(* Logix 5000 project; controller PBS_Perfusion vendor 1 type 14 code 217 rev 32.14; software revision 32.03; part 25 of 27 *)
(* tags used below, declared in another part *)
   AIC703 : P_AInAdv;   // BRX DO PV
   AT701 : P_AInAdv;   // DO Transmitter
   AT702 : P_AInAdv;   // pH Transmitter
   BRX_Comm_Toggle : BOOL;
   BRX_Data : PBSdata_UDT;
   Brx_heartbeat_Alarm : BOOL;
   Brx_Heartbeat_Alarm_Reset : BOOL;
   BRX_Heartbeat_Fail : TIMER;
   BRX_HiAdj : BOOL;   // BRX HI adj in progress
   BRX_HiAdjEnable : BOOL;
   BRX_HiAdjTimer : TIMER;
   BRX_HiadjTimeSP : REAL;
   BRX_HiSP : REAL;
   BRX_LoAdj : BOOL;   // BRX Lo Adj in progress
   BRX_LoAdjEnable : BOOL;
   BRX_LoAdjTimer : TIMER;
   BRX_LoadjTimeSP : REAL;
   BRX_LoSP : REAL;
   ConditionedMedia_Initialize : BOOL;
   ConditionedMedia_Scaler : SCALE;
   CondMed_AdjustInProgress : BOOL;
   EStop : P_DIn;
   Heater_Output : P_AOut;   // Heating blanket AO
   Heater_Output_intlk : P_Intlk;
   Json_Alarm : BOOL;
   LIT801 : P_AInAdv;   // Level Value From BRX
   MCV_HiAdj : BOOL;   // MCV hi adjust active
   MCV_HiAdjEnable : BOOL;
   MCV_HiAdjTimer : TIMER;
   MCV_HiAdjTimeSP : REAL;
   MCV_HiSP : REAL;
   ONS : DINT[3];
   P101 : P_VSD;   // Feed Pump
   P101_Alarm_Reset : AMP_Alarm_Reset;
   P101_Cal : Pump_Cal;
   P101_Cal_Constant : REAL;
   P101_Crash_Stop : AMP_Crash_Stop;
   P101_Dose_Running : BOOL;
   P101_Dose_Speed_mlmin : REAL;
   P101_Enable : AMP_Motor_Enable;
   P101_FaultCodeList : P_DescList[1];
   P101_Input_Assembly : AMP_Input_Assembly_v2;
   P101_Input_Assembly_Instance : AMP_Input_Assembly;
   P101_intlk : P_Intlk;
   P101_Jog_Move : AMP_Jog_Move;
   P101_Relative_Move : AMP_Relative_Move;
   P101_Status_Code : AMP_Status_Code;
   P101_Update_Jog_Speed : AMP_Update_Jog_Speed;
   P101Fault : BOOL;
   P101Fault_Output : BOOL;
   P102 : P_VSD;   // Media Pump
   P102_Alarm_Reset : AMP_Alarm_Reset;
   P102_Cal : Pump_Cal;
   P102_Cal_Constant : REAL;
   P102_Crash_Stop : AMP_Crash_Stop;
   P102_Enable : AMP_Motor_Enable;
   P102_FaultCodeList : P_DescList[1];
   P102_Input_Assembly : AMP_Input_Assembly_v2;
   P102_Input_Assembly_Instance : AMP_Input_Assembly;
   P102_intlk : P_Intlk;
   P102_Jog_Move : AMP_Jog_Move;
   P102_Relative_Move : AMP_Relative_Move;
   P102_Status_Code : AMP_Status_Code;
   P102_Update_Jog_Speed : AMP_Update_Jog_Speed;
   P103 : P_VSD;   // Conditioned Media Addition Pump
   P103_Alarm_Reset : AMP_Alarm_Reset;
   P103_Cal : Pump_Cal;
   P103_Cal_Constant : REAL;
   P103_Crash_Stop : AMP_Crash_Stop;
   P103_Enable : AMP_Motor_Enable;
   P103_FaultCodeList : P_DescList[1];
   P103_Input_Assembly : AMP_Input_Assembly_v2;
   P103_Input_Assembly_Instance : AMP_Input_Assembly;
   P103_intlk : P_Intlk;
   P103_Jog_Move : AMP_Jog_Move;
   P103_Relative_Move : AMP_Relative_Move;
   P103_Status_Code : AMP_Status_Code;
   P103_Update_Jog_Speed : AMP_Update_Jog_Speed;
   P104 : P_VSD;   // Recirculation Pump
   P104_Alarm_Reset : AMP_Alarm_Reset;
   P104_Cal : Pump_Cal;
   P104_Cal_Constant : REAL;
   P104_Crash_Stop : AMP_Crash_Stop;
   P104_Enable : AMP_Motor_Enable;
   P104_FaultCodeList : P_DescList[1];
   P104_Input_Assembly : AMP_Input_Assembly_v2;
   P104_Input_Assembly_Instance : AMP_Input_Assembly;
   p104_intlk : P_Intlk;
   P104_Jog_Move : AMP_Jog_Move;
   P104_Relative_Move : AMP_Relative_Move;
   P104_Status_Code : AMP_Status_Code;
   P104_Update_Jog_Speed : AMP_Update_Jog_Speed;
   P105 : P_VSD;   // Spent Media Pump
   P105_FaultCodeList : P_DescList[1];
   P105_intlk : P_Intlk;
   Recirc_HiSP1 : REAL;   // BRX Hi recirc hi speed modifier
   Recirc_LoSP1 : REAL;   // MCV Hi recirc lo speed modifier
   Recirc_LoSP2 : REAL;   // BRX Lo recirc lo speed modifier
   SIC401 : P_VSD;   // Agitator
   SIC401_FaultCodeList : P_DescList[1];   // made for agaitor p_VSD block
   SIC401_intlk : P_Intlk;
   Temp_Limit_Adm : REAL;
   Temp_Scaler : SCALE;
   Test_Temp_Raw : REAL;
   TT700 : P_AInAdv;   // Temperature Transmitter
   WT701 : P_AInAdv;   // Media Scale
   WT702 : P_AInAdv;   // MCV Weight
   WT703 : P_AInAdv;   // Spent Media/Harvest Scale

PROGRAM CM_PBS   (* main routine Main *)
VAR
   BOR_01 : FBD_BOOLEAN_OR;
   SEL_01 : SELECT := (In2 := 200.0);
   TOT_01 : TOTALIZER := (Gain := 1.0, RTSTime := 1);
   TOT_02 : TOTALIZER := (Gain := 1.0, RTSTime := 1);
END_VAR

ROUTINE Brx_Comms   (* ladder *)
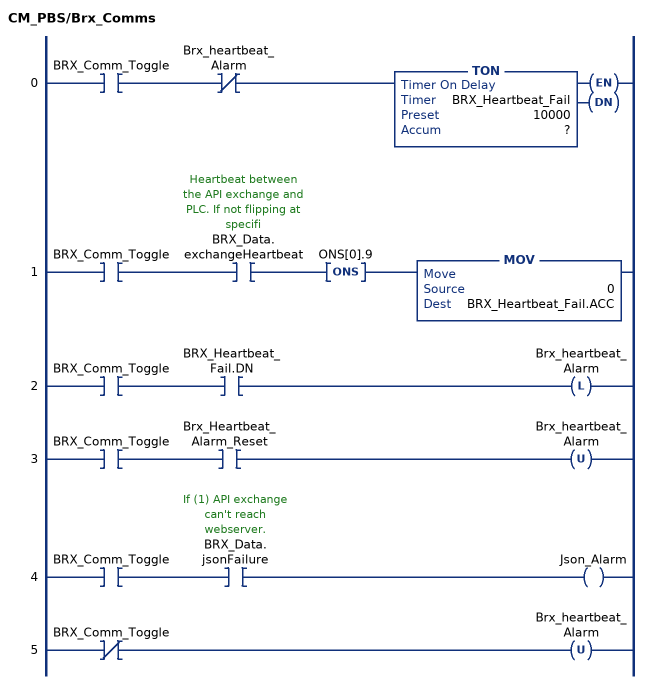
   0: XIC(BRX_Comm_Toggle)XIO(Brx_heartbeat_Alarm)TON(BRX_Heartbeat_Fail,?,?);
   1: XIC(BRX_Comm_Toggle)XIC(BRX_Data.exchangeHeartbeat)ONS(ONS[0].9)MOV(0,BRX_Heartbeat_Fail.ACC);
   2: XIC(BRX_Comm_Toggle)XIC(BRX_Heartbeat_Fail.DN)OTL(Brx_heartbeat_Alarm);
   3: XIC(BRX_Comm_Toggle)XIC(Brx_Heartbeat_Alarm_Reset)OTU(Brx_heartbeat_Alarm);
   4: XIC(BRX_Comm_Toggle)XIC(BRX_Data.jsonFailure)OTE(Json_Alarm);
   5: XIO(BRX_Comm_Toggle)OTU(Brx_heartbeat_Alarm);
END_ROUTINE

ROUTINE CM_Agitator   (* ladder *)
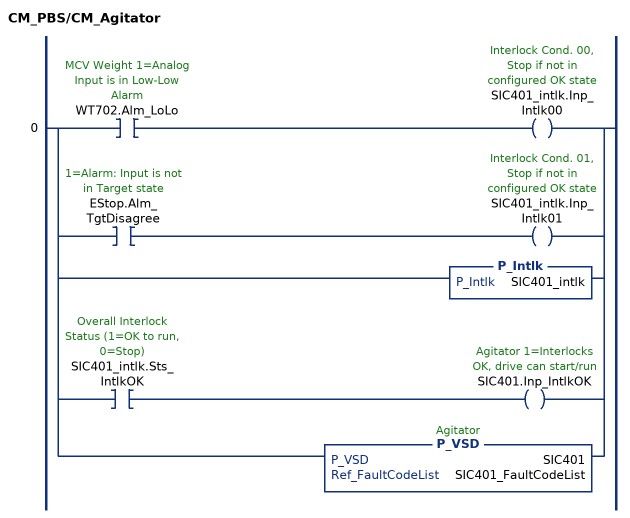
   0: [[XIC(WT702.Alm_LoLo) OTE(SIC401_intlk.Inp_Intlk00) ,XIC(EStop.Alm_TgtDisagree) OTE(SIC401_intlk.Inp_Intlk01) ,P_Intlk(SIC401_intlk) ,XIC(SIC401_intlk.Sts_IntlkOK) OTE(SIC401.Inp_IntlkOK) ] ,P_VSD(SIC401,SIC401_FaultCodeList) ];
END_ROUTINE

ROUTINE CM_AI   (* ladder *)
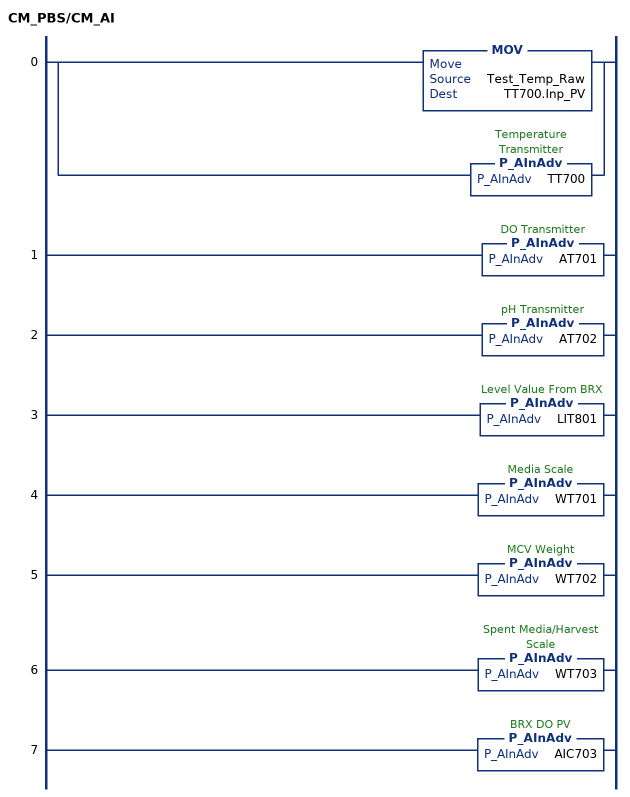
   0: [MOV(Test_Temp_Raw,TT700.Inp_PV) ,P_AInAdv(TT700) ];
   1: P_AInAdv(AT701);
   2: P_AInAdv(AT702);
   3: P_AInAdv(LIT801);
   4: P_AInAdv(WT701);
   5: P_AInAdv(WT702);
   6: P_AInAdv(WT703);
   7: P_AInAdv(AIC703);
END_ROUTINE

ROUTINE CM_AO   (* ladder *)
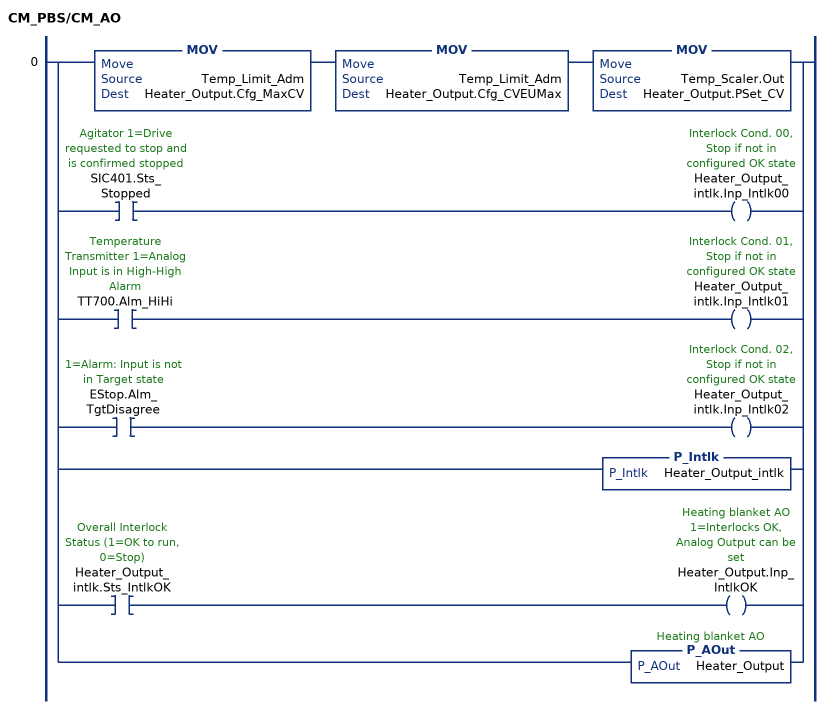
   0: [MOV(Temp_Limit_Adm,Heater_Output.Cfg_MaxCV) MOV(Temp_Limit_Adm,Heater_Output.Cfg_CVEUMax) MOV(Temp_Scaler.Out,Heater_Output.PSet_CV) ,[XIC(SIC401.Sts_Stopped) OTE(Heater_Output_intlk.Inp_Intlk00) ,XIC(TT700.Alm_HiHi) OTE(Heater_Output_intlk.Inp_Intlk01) ,XIC(EStop.Alm_TgtDisagree) OTE(Heater_Output_intlk.Inp_Intlk02) ,P_Intlk(Heater_Output_intlk) ,XIC(Heater_Output_intlk.Sts_IntlkOK) OTE(Heater_Output.Inp_IntlkOK) ] ,P_AOut(Heater_Output) ];
END_ROUTINE

ROUTINE CM_DI   (* ladder *)
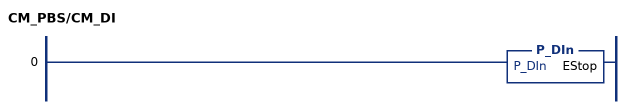
   0: P_DIn(EStop);
END_ROUTINE

ROUTINE CM_DO   (* ladder *)
END_ROUTINE

ROUTINE CM_Pumps   (* ladder *)
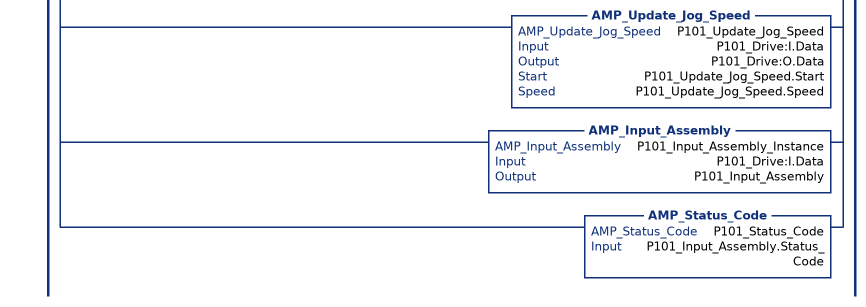
   0: [XIC(P101Fault) OTE(P101Fault_Output) ,[XIC(LIT801.Alm_HiHi) OTE(P101_intlk.Inp_Intlk00) ,XIC(WT701.Alm_LoLo) OTE(P101_intlk.Inp_Intlk01) ,XIC(EStop.Alm_TgtDisagree) OTE(P101_intlk.Inp_Intlk02) ,P_Intlk(P101_intlk) ,XIC(P101_intlk.Sts_IntlkOK) OTE(P101.Inp_IntlkOK) ] ,[P_VSD(P101,P101_FaultCodeList) ,XIC(P101.Sts_StartingFwd) OTL(P101_Jog_Move.Start) ,XIC(P101.Sts_StoppingFwd) OTL(P101_Crash_Stop.Stop) ,XIC(P101_Status_Code.Moving) OTU(P101_Jog_Move.Start) ,XIO(P101_Status_Code.Moving) OTU(P101_Crash_Stop.Stop) ,CPT(P101_Jog_Move.Speed,P101.Val_SpeedRef/ ( P101_Cal_Constant * 60)) ,NEQ(P101_Update_Jog_Speed.Speed,P101_Jog_Move.Speed) ONS(ONS[0].5) MOV(P101_Jog_Move.Speed,P101_Update_Jog_Speed.Speed) OTE(P101_Update_Jog_Speed.Start) ] ,AFI() Pump_Cal(P101_Cal,P101.Sts_RunningFwd,P101.PCmd_Prog,P101.Cfg_SpeedRefEUMin,P101.Cfg_SpeedRefEUMax,P101.Cfg_SpeedFdbkEUMin,P101.Cfg_SpeedFdbkEUMax,P101.Cfg_MinSpdRef,P101.Cfg_MaxSpdRef,P101.PSet_SpeedRef,P101.PCmd_StartFwd,P101.Sts_Prog,P101.PCmd_Stop) ,AMP_Motor_Enable(P101_Enable,P101_Drive:I.Data,P101_Drive:O.Data,P101_Enable.Enable) ,AMP_Alarm_Reset(P101_Alarm_Reset,P101_Drive:I.Data,P101_Drive:O.Data,P101_Alarm_Reset.Reset) ,AMP_Jog_Move(P101_Jog_Move,P101_Drive:I.Data,P101_Drive:O.Data,P101_Jog_Move.Start,P101_Jog_Move.Speed,P101_Jog_Move.Acc,P101_Jog_Move.Dec) ,AMP_Crash_Stop(P101_Crash_Stop,P101_Drive:I.Data,P101_Drive:O.Data,P101_Crash_Stop.Stop) ,AMP_Relative_Move(P101_Relative_Move,P101_Drive:I.Data,P101_Drive:O.Data,P101_Relative_Move.Start,P101_Relative_Move.Distance,P101_Relative_Move.Speed,P101_Relative_Move.Acc,P101_Relative_Move.Dec) ,AMP_Update_Jog_Speed(P101_Update_Jog_Speed,P101_Drive:I.Data,P101_Drive:O.Data,P101_Update_Jog_Speed.Start,P101_Update_Jog_Speed.Speed) ,AMP_Input_Assembly(P101_Input_Assembly_Instance,P101_Drive:I.Data,P101_Input_Assembly) ,AMP_Status_Code(P101_Status_Code,P101_Input_Assembly.Status_Code) ];
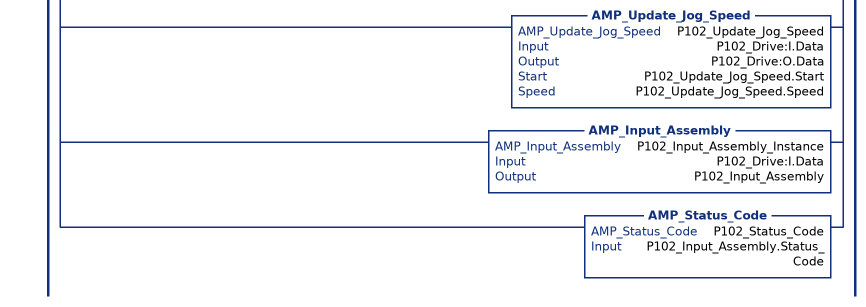
   1: [[XIC(WT702.Alm_HiHi) OTE(P102_intlk.Inp_Intlk00) ,XIC(WT701.Alm_LoLo) OTE(P102_intlk.Inp_Intlk01) ,XIC(EStop.Alm_TgtDisagree) OTE(P102_intlk.Inp_Intlk02) ,P_Intlk(P102_intlk) ,XIC(P102_intlk.Sts_IntlkOK) OTE(P102.Inp_IntlkOK) ] ,[P_VSD(P102,P102_FaultCodeList) ,XIC(P102.Sts_StartingFwd) OTL(P102_Jog_Move.Start) ,XIC(P102.Sts_StoppingFwd) OTL(P102_Crash_Stop.Stop) ,XIC(P102_Status_Code.Moving) OTU(P102_Jog_Move.Start) ,XIO(P102_Status_Code.Moving) OTU(P102_Crash_Stop.Stop) ,CPT(P102_Jog_Move.Speed,P102.Val_SpeedRef/ ( P102_Cal_Constant * 60)) ,NEQ(P102_Update_Jog_Speed.Speed,P102_Jog_Move.Speed) ONS(ONS[0].5) MOV(P102_Jog_Move.Speed,P102_Update_Jog_Speed.Speed) OTE(P102_Update_Jog_Speed.Start) ] ,AFI() Pump_Cal(P102_Cal,P102.Sts_RunningFwd,P102.PCmd_Prog,P102.Cfg_SpeedRefEUMin,P102.Cfg_SpeedRefEUMax,P102.Cfg_SpeedFdbkEUMin,P102.Cfg_SpeedFdbkEUMax,P102.Cfg_MinSpdRef,P102.Cfg_MaxSpdRef,P102.PSet_SpeedRef,P102.PCmd_StartFwd,P102.Sts_Prog,P102.PCmd_Stop) ,AMP_Motor_Enable(P102_Enable,P102_Drive:I.Data,P102_Drive:O.Data,P102_Enable.Enable) ,AMP_Alarm_Reset(P102_Alarm_Reset,P102_Drive:I.Data,P102_Drive:O.Data,P102_Alarm_Reset.Reset) ,AMP_Jog_Move(P102_Jog_Move,P102_Drive:I.Data,P102_Drive:O.Data,P102_Jog_Move.Start,P102_Jog_Move.Speed,P102_Jog_Move.Acc,P102_Jog_Move.Dec) ,AMP_Crash_Stop(P102_Crash_Stop,P102_Drive:I.Data,P102_Drive:O.Data,P102_Crash_Stop.Stop) ,AMP_Relative_Move(P102_Relative_Move,P102_Drive:I.Data,P102_Drive:O.Data,P102_Relative_Move.Start,P102_Relative_Move.Distance,P102_Relative_Move.Speed,P102_Relative_Move.Acc,P102_Relative_Move.Dec) ,AMP_Update_Jog_Speed(P102_Update_Jog_Speed,P102_Drive:I.Data,P102_Drive:O.Data,P102_Update_Jog_Speed.Start,P102_Update_Jog_Speed.Speed) ,AMP_Input_Assembly(P102_Input_Assembly_Instance,P102_Drive:I.Data,P102_Input_Assembly) ,AMP_Status_Code(P102_Status_Code,P102_Input_Assembly.Status_Code) ];
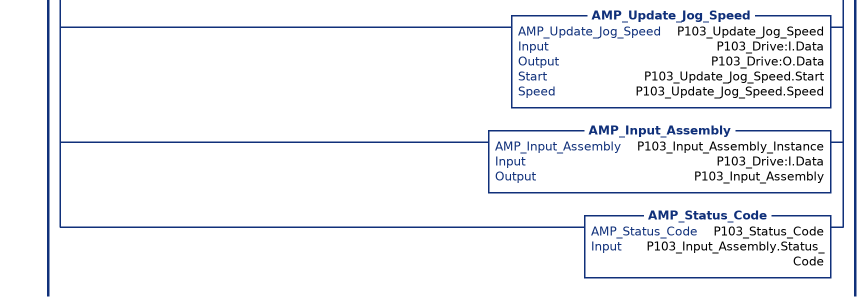
   2: [[XIC(LIT801.Alm_HiHi) OTE(P103_intlk.Inp_Intlk00) ,XIC(WT702.Alm_LoLo) OTE(P103_intlk.Inp_Intlk01) ,XIC(EStop.Alm_TgtDisagree) OTE(P103_intlk.Inp_Intlk02) ,P_Intlk(P103_intlk) ,XIC(P103_intlk.Sts_IntlkOK) OTE(P103.Inp_IntlkOK) ] ,[P_VSD(P103,P103_FaultCodeList) ,XIC(P103.Sts_StartingFwd) OTL(P103_Jog_Move.Start) ,XIC(P103.Sts_StoppingFwd) OTL(P103_Crash_Stop.Stop) ,XIC(P103_Status_Code.Moving) OTU(P103_Jog_Move.Start) ,XIO(P103_Status_Code.Moving) OTU(P103_Crash_Stop.Stop) ,CPT(P103_Jog_Move.Speed,P103.Val_SpeedRef/ ( P103_Cal_Constant * 60)) ,NEQ(P103_Update_Jog_Speed.Speed,P103_Jog_Move.Speed) ONS(ONS[0].5) MOV(P103_Jog_Move.Speed,P103_Update_Jog_Speed.Speed) OTE(P102_Update_Jog_Speed.Start) ] ,AFI() Pump_Cal(P103_Cal,P103.Sts_RunningFwd,P103.PCmd_Prog,P103.Cfg_SpeedRefEUMin,P103.Cfg_SpeedRefEUMax,P103.Cfg_SpeedFdbkEUMin,P103.Cfg_SpeedFdbkEUMax,P103.Cfg_MinSpdRef,P103.Cfg_MaxSpdRef,P103.PSet_SpeedRef,P103.PCmd_StartFwd,P103.Sts_Prog,P103.PCmd_Stop) ,AMP_Motor_Enable(P103_Enable,P103_Drive:I.Data,P103_Drive:O.Data,P103_Enable.Enable) ,AMP_Alarm_Reset(P103_Alarm_Reset,P103_Drive:I.Data,P103_Drive:O.Data,P103_Alarm_Reset.Reset) ,AMP_Jog_Move(P103_Jog_Move,P103_Drive:I.Data,P103_Drive:O.Data,P103_Jog_Move.Start,P103_Jog_Move.Speed,P103_Jog_Move.Acc,P103_Jog_Move.Dec) ,AMP_Crash_Stop(P103_Crash_Stop,P103_Drive:I.Data,P103_Drive:O.Data,P103_Crash_Stop.Stop) ,AMP_Relative_Move(P103_Relative_Move,P103_Drive:I.Data,P103_Drive:O.Data,P103_Relative_Move.Start,P103_Relative_Move.Distance,P103_Relative_Move.Speed,P103_Relative_Move.Acc,P103_Relative_Move.Dec) ,AMP_Update_Jog_Speed(P103_Update_Jog_Speed,P103_Drive:I.Data,P103_Drive:O.Data,P103_Update_Jog_Speed.Start,P103_Update_Jog_Speed.Speed) ,AMP_Input_Assembly(P103_Input_Assembly_Instance,P103_Drive:I.Data,P103_Input_Assembly) ,AMP_Status_Code(P103_Status_Code,P103_Input_Assembly.Status_Code) ];
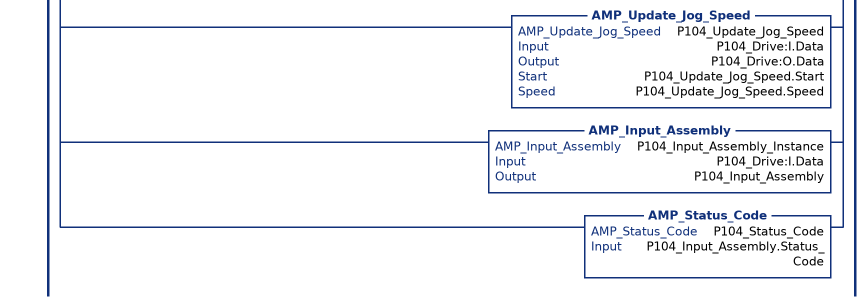
   3: [[XIC(LIT801.Alm_LoLo) OTE(p104_intlk.Inp_Intlk00) ,XIC(WT702.Alm_HiHi) OTE(p104_intlk.Inp_Intlk01) ,XIC(EStop.Alm_TgtDisagree) OTE(p104_intlk.Inp_Intlk02) ,P_Intlk(p104_intlk) ,XIC(p104_intlk.Sts_IntlkOK) OTE(P104.Inp_IntlkOK) ] ,[P_VSD(P104,P104_FaultCodeList) ,XIC(P104.Sts_StartingFwd) OTL(P104_Jog_Move.Start) ,XIC(P104.Sts_StoppingFwd) OTL(P104_Crash_Stop.Stop) ,XIC(P104_Status_Code.Moving) OTU(P104_Jog_Move.Start) ,XIO(P104_Status_Code.Moving) OTU(P104_Crash_Stop.Stop) ,CPT(P104_Jog_Move.Speed,P104.Val_SpeedRef/ ( P104_Cal_Constant * 60)) ,NEQ(P104_Update_Jog_Speed.Speed,P104_Jog_Move.Speed) ONS(ONS[0].5) MOV(P104_Jog_Move.Speed,P104_Update_Jog_Speed.Speed) OTE(P104_Update_Jog_Speed.Start) ] ,AFI() Pump_Cal(P104_Cal,P104.Sts_RunningFwd,P104.PCmd_Prog,P104.Cfg_SpeedRefEUMin,P104.Cfg_SpeedRefEUMax,P104.Cfg_SpeedFdbkEUMin,P104.Cfg_SpeedFdbkEUMax,P104.Cfg_MinSpdRef,P104.Cfg_MaxSpdRef,P104.PSet_SpeedRef,P104.PCmd_StartFwd,P104.Sts_Prog,P104.PCmd_Stop) ,AMP_Motor_Enable(P104_Enable,P104_Drive:I.Data,P104_Drive:O.Data,P104_Enable.Enable) ,AMP_Alarm_Reset(P104_Alarm_Reset,P104_Drive:I.Data,P104_Drive:O.Data,P104_Alarm_Reset.Reset) ,AMP_Jog_Move(P104_Jog_Move,P104_Drive:I.Data,P104_Drive:O.Data,P104_Jog_Move.Start,P104_Jog_Move.Speed,P104_Jog_Move.Acc,P104_Jog_Move.Dec) ,AMP_Crash_Stop(P104_Crash_Stop,P104_Drive:I.Data,P104_Drive:O.Data,P104_Crash_Stop.Stop) ,AMP_Relative_Move(P104_Relative_Move,P104_Drive:I.Data,P104_Drive:O.Data,P104_Relative_Move.Start,P104_Relative_Move.Distance,P104_Relative_Move.Speed,P104_Relative_Move.Acc,P104_Relative_Move.Dec) ,AMP_Update_Jog_Speed(P104_Update_Jog_Speed,P104_Drive:I.Data,P104_Drive:O.Data,P104_Update_Jog_Speed.Start,P104_Update_Jog_Speed.Speed) ,AMP_Input_Assembly(P104_Input_Assembly_Instance,P104_Drive:I.Data,P104_Input_Assembly) ,AMP_Status_Code(P104_Status_Code,P104_Input_Assembly.Status_Code) ];
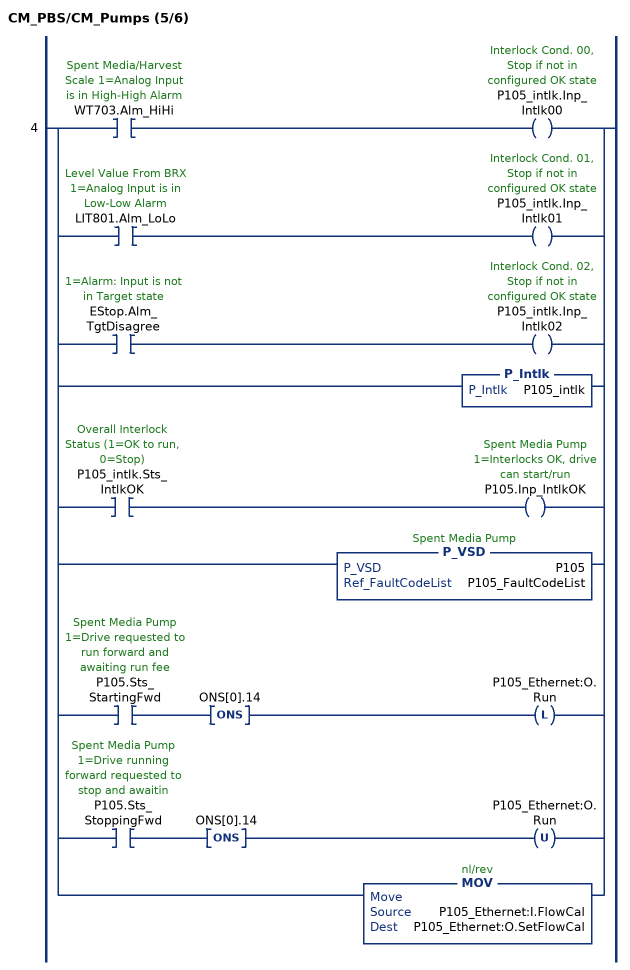
   4 (stored rung type 14): [[XIC(WT703.Alm_HiHi) OTE(P105_intlk.Inp_Intlk00) ,XIC(LIT801.Alm_LoLo) OTE(P105_intlk.Inp_Intlk01) ,XIC(EStop.Alm_TgtDisagree) OTE(P105_intlk.Inp_Intlk02) ,P_Intlk(P105_intlk) ,XIC(P105_intlk.Sts_IntlkOK) OTE(P105.Inp_IntlkOK) ] ,P_VSD(P105,P105_FaultCodeList) ,XIC(P105.Sts_StartingFwd) ONS(ONS[0].14) OTL(P105_Ethernet:O.Run) ,XIC(P105.Sts_StoppingFwd) ONS(ONS[0].14) OTU(P105_Ethernet:O.Run) ,MOV(P105_Ethernet:I.FlowCal,P105_Ethernet:O.SetFlowCal) ];
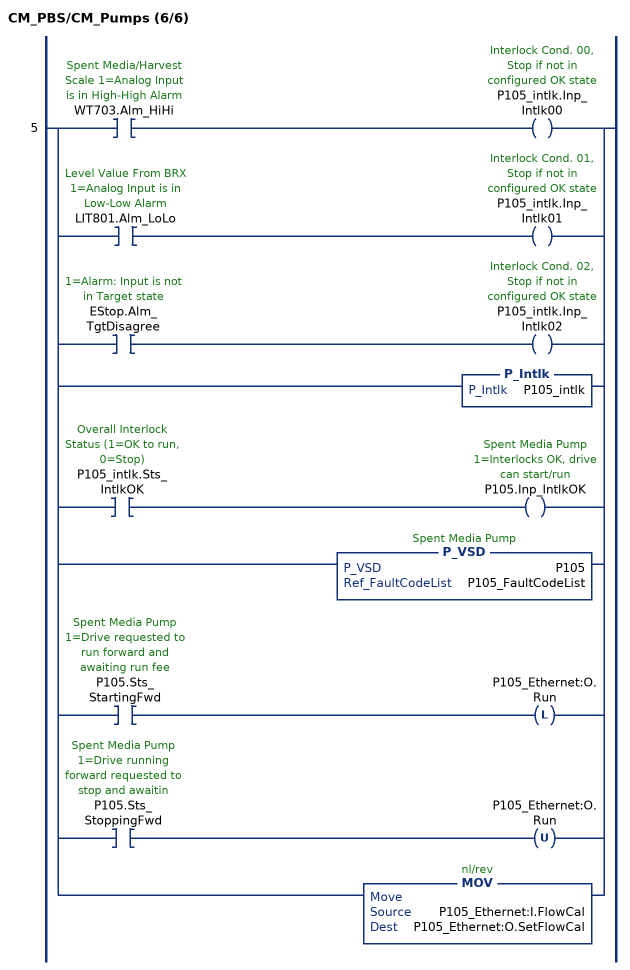
   5 (stored rung type 10): [[XIC(WT703.Alm_HiHi) OTE(P105_intlk.Inp_Intlk00) ,XIC(LIT801.Alm_LoLo) OTE(P105_intlk.Inp_Intlk01) ,XIC(EStop.Alm_TgtDisagree) OTE(P105_intlk.Inp_Intlk02) ,P_Intlk(P105_intlk) ,XIC(P105_intlk.Sts_IntlkOK) OTE(P105.Inp_IntlkOK) ] ,P_VSD(P105,P105_FaultCodeList) ,XIC(P105.Sts_StartingFwd) OTL(P105_Ethernet:O.Run) ,XIC(P105.Sts_StoppingFwd) OTU(P105_Ethernet:O.Run) ,MOV(P105_Ethernet:I.FlowCal,P105_Ethernet:O.SetFlowCal) ];
END_ROUTINE

ROUTINE CM_Totalizers   (* function block diagram *)
// Totalizers
   SHEET 1
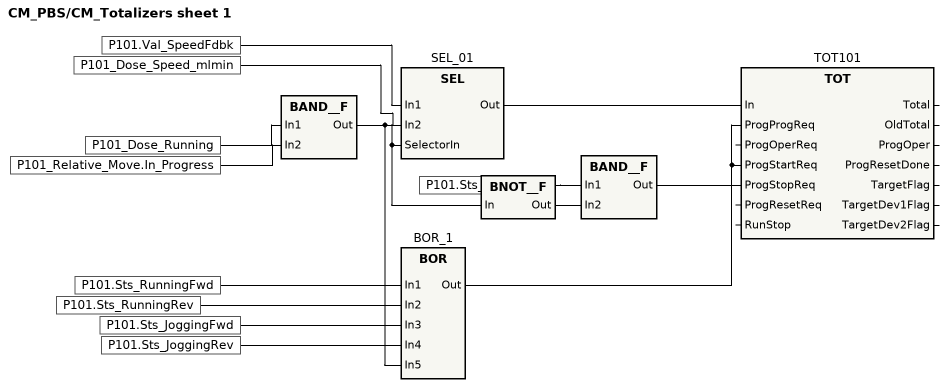
   BAND__F_1 : BAND__F(In1 := P101_Dose_Running, In2 := P101_Relative_Move.In_Progress);
   SEL_01 : SEL(In1 := P101.Val_SpeedFdbk, In2 := P101_Dose_Speed_mlmin, SelectorIn := BAND__F_1.Out);
   BOR_1 : BOR(In1 := P101.Sts_RunningFwd, In2 := P101.Sts_RunningRev, In3 := P101.Sts_JoggingFwd, In4 := P101.Sts_JoggingRev, In5 := BAND__F_1.Out);
   BNOT__F_2 : BNOT__F(In := BAND__F_1.Out);
   BAND__F_3 : BAND__F(In1 := P101.Sts_Stopped, In2 := BNOT__F_2.Out);
   TOT101 : TOT(In := SEL_01.Out, ProgProgReq := BOR_1.Out, ProgStartReq := BOR_1.Out, ProgStopReq := BAND__F_3.Out);   // unwired pins: ProgOperReq ProgResetReq Total OldTotal ProgOper RunStop ProgResetDone TargetFlag TargetDev1Flag TargetDev2Flag
   SHEET 2
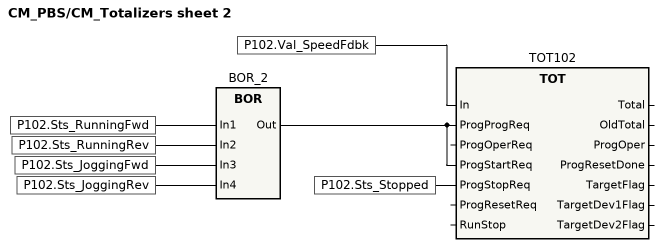
   BOR_2 : BOR(In1 := P102.Sts_RunningFwd, In2 := P102.Sts_RunningRev, In3 := P102.Sts_JoggingFwd, In4 := P102.Sts_JoggingRev);
   TOT102 : TOT(In := P102.Val_SpeedFdbk, ProgProgReq := BOR_2.Out, ProgStartReq := BOR_2.Out, ProgStopReq := P102.Sts_Stopped);   // unwired pins: ProgOperReq ProgResetReq Total OldTotal ProgOper RunStop ProgResetDone TargetFlag TargetDev1Flag TargetDev2Flag
   SHEET 3
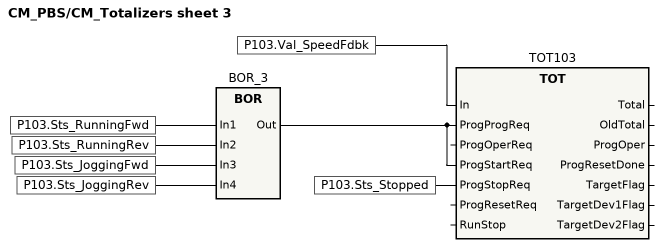
   BOR_3 : BOR(In1 := P103.Sts_RunningFwd, In2 := P103.Sts_RunningRev, In3 := P103.Sts_JoggingFwd, In4 := P103.Sts_JoggingRev);
   TOT103 : TOT(In := P103.Val_SpeedFdbk, ProgProgReq := BOR_3.Out, ProgStartReq := BOR_3.Out, ProgStopReq := P103.Sts_Stopped);   // unwired pins: ProgOperReq ProgResetReq Total OldTotal ProgOper RunStop ProgResetDone TargetFlag TargetDev1Flag TargetDev2Flag
   SHEET 4
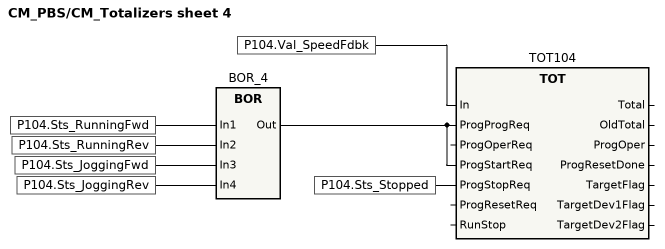
   BOR_4 : BOR(In1 := P104.Sts_RunningFwd, In2 := P104.Sts_RunningRev, In3 := P104.Sts_JoggingFwd, In4 := P104.Sts_JoggingRev);
   TOT104 : TOT(In := P104.Val_SpeedFdbk, ProgProgReq := BOR_4.Out, ProgStartReq := BOR_4.Out, ProgStopReq := P104.Sts_Stopped);   // unwired pins: ProgOperReq ProgResetReq Total OldTotal ProgOper RunStop ProgResetDone TargetFlag TargetDev1Flag TargetDev2Flag
   SHEET 5
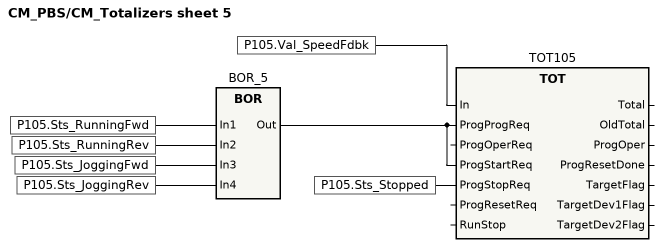
   BOR_5 : BOR(In1 := P105.Sts_RunningFwd, In2 := P105.Sts_RunningRev, In3 := P105.Sts_JoggingFwd, In4 := P105.Sts_JoggingRev);
   TOT105 : TOT(In := P105.Val_SpeedFdbk, ProgProgReq := BOR_5.Out, ProgStartReq := BOR_5.Out, ProgStopReq := P105.Sts_Stopped);   // unwired pins: ProgOperReq ProgResetReq Total OldTotal ProgOper RunStop ProgResetDone TargetFlag TargetDev1Flag TargetDev2Flag
END_ROUTINE

ROUTINE Conditioned_Addition_Control   (* ladder *)
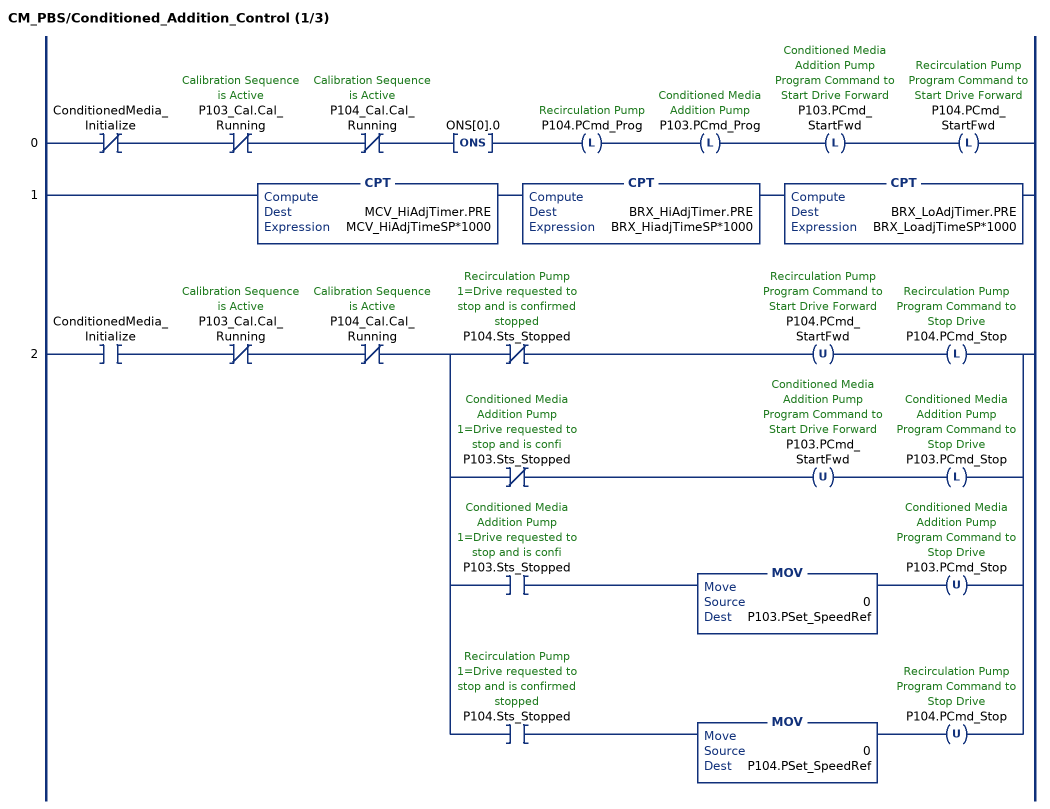
   0: XIO(ConditionedMedia_Initialize)XIO(P103_Cal.Cal_Running)XIO(P104_Cal.Cal_Running)ONS(ONS[0].0)OTL(P104.PCmd_Prog)OTL(P103.PCmd_Prog)OTL(P103.PCmd_StartFwd)OTL(P104.PCmd_StartFwd);
   1: CPT(MCV_HiAdjTimer.PRE,MCV_HiAdjTimeSP*1000)CPT(BRX_HiAdjTimer.PRE,BRX_HiadjTimeSP*1000)CPT(BRX_LoAdjTimer.PRE,BRX_LoadjTimeSP*1000);
   2: XIC(ConditionedMedia_Initialize)XIO(P103_Cal.Cal_Running)XIO(P104_Cal.Cal_Running)[XIO(P104.Sts_Stopped) OTU(P104.PCmd_StartFwd) OTL(P104.PCmd_Stop) ,XIO(P103.Sts_Stopped) OTU(P103.PCmd_StartFwd) OTL(P103.PCmd_Stop) ,XIC(P103.Sts_Stopped) MOV(0,P103.PSet_SpeedRef) OTU(P103.PCmd_Stop) ,XIC(P104.Sts_Stopped) MOV(0,P104.PSet_SpeedRef) OTU(P104.PCmd_Stop) ];
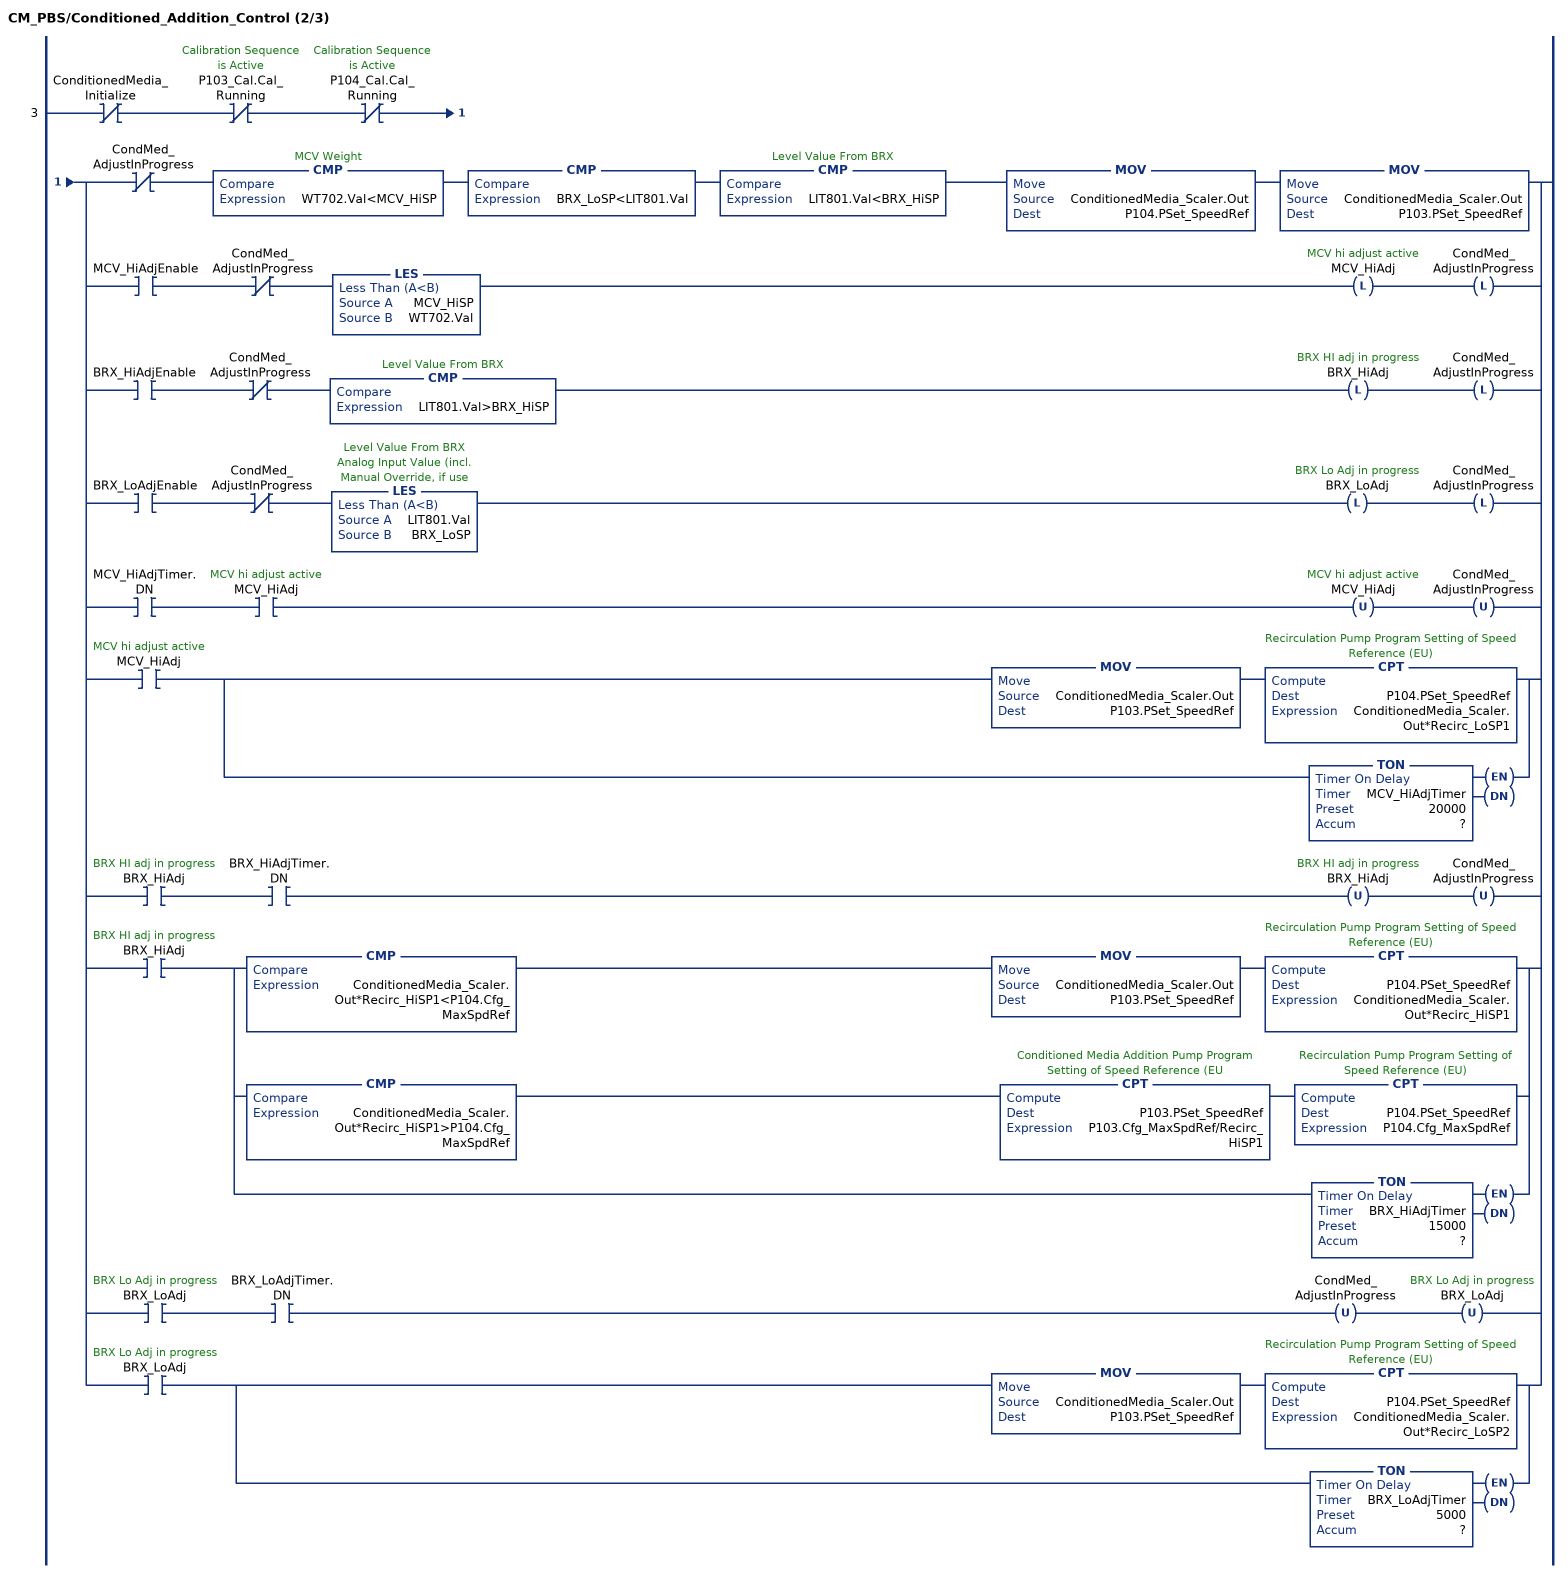
   3: XIO(ConditionedMedia_Initialize)XIO(P103_Cal.Cal_Running)XIO(P104_Cal.Cal_Running)[XIO(CondMed_AdjustInProgress) CMP(WT702.Val<MCV_HiSP) CMP(BRX_LoSP<LIT801.Val) CMP(LIT801.Val<BRX_HiSP) MOV(ConditionedMedia_Scaler.Out,P104.PSet_SpeedRef) MOV(ConditionedMedia_Scaler.Out,P103.PSet_SpeedRef) ,XIC(MCV_HiAdjEnable) XIO(CondMed_AdjustInProgress) LES(MCV_HiSP,WT702.Val) OTL(MCV_HiAdj) OTL(CondMed_AdjustInProgress) ,XIC(BRX_HiAdjEnable) XIO(CondMed_AdjustInProgress) CMP(LIT801.Val>BRX_HiSP) OTL(BRX_HiAdj) OTL(CondMed_AdjustInProgress) ,XIC(BRX_LoAdjEnable) XIO(CondMed_AdjustInProgress) LES(LIT801.Val,BRX_LoSP) OTL(BRX_LoAdj) OTL(CondMed_AdjustInProgress) ,XIC(MCV_HiAdjTimer.DN) XIC(MCV_HiAdj) OTU(MCV_HiAdj) OTU(CondMed_AdjustInProgress) ,XIC(MCV_HiAdj) [MOV(ConditionedMedia_Scaler.Out,P103.PSet_SpeedRef) CPT(P104.PSet_SpeedRef,ConditionedMedia_Scaler.Out*Recirc_LoSP1) ,TON(MCV_HiAdjTimer,?,?) ] ,XIC(BRX_HiAdj) XIC(BRX_HiAdjTimer.DN) OTU(BRX_HiAdj) OTU(CondMed_AdjustInProgress) ,XIC(BRX_HiAdj) [CMP(ConditionedMedia_Scaler.Out*Recirc_HiSP1<P104.Cfg_MaxSpdRef) MOV(ConditionedMedia_Scaler.Out,P103.PSet_SpeedRef) CPT(P104.PSet_SpeedRef,ConditionedMedia_Scaler.Out*Recirc_HiSP1) ,CMP(ConditionedMedia_Scaler.Out*Recirc_HiSP1>P104.Cfg_MaxSpdRef) CPT(P103.PSet_SpeedRef,P103.Cfg_MaxSpdRef/Recirc_HiSP1) CPT(P104.PSet_SpeedRef,P104.Cfg_MaxSpdRef) ,TON(BRX_HiAdjTimer,?,?) ] ,XIC(BRX_LoAdj) XIC(BRX_LoAdjTimer.DN) OTU(CondMed_AdjustInProgress) OTU(BRX_LoAdj) ,XIC(BRX_LoAdj) [MOV(ConditionedMedia_Scaler.Out,P103.PSet_SpeedRef) CPT(P104.PSet_SpeedRef,ConditionedMedia_Scaler.Out*Recirc_LoSP2) ,TON(BRX_LoAdjTimer,?,?) ] ];
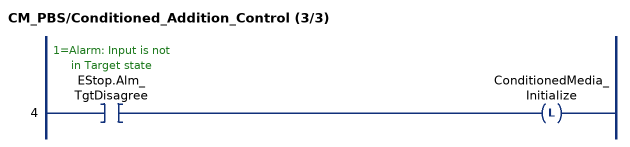
   4: XIC(EStop.Alm_TgtDisagree)OTL(ConditionedMedia_Initialize);
END_ROUTINE
